{attribute 'qualified_only'}
VAR_GLOBAL
	//cmActuator2State : Udt_CM_Actuator2State;
	Udt_PlantControl : Udt_PlantControl;
END_VAR

(* stored: Version 1.1.0.1, ProductVersion 3.1.4024.13
   GVL OPC: Id {e0cd9ffc-1253-4fa9-9b6c-11bdc95bd4be} *)
